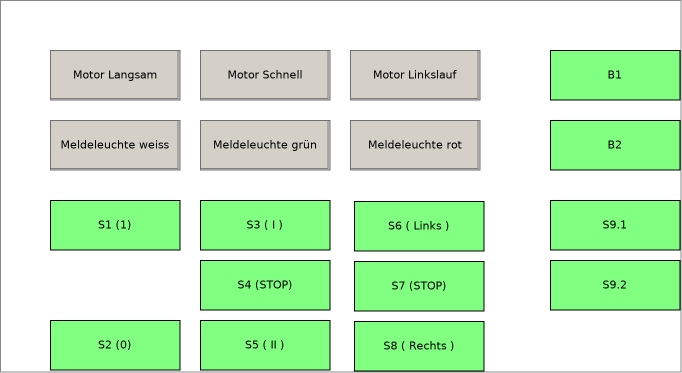
VISUALIZATION VisuGetriebemotor  // 682x373
    Button (50,50 130x50), "Motor Langsam"
        tap dSub.Q3
    Button (200,50 130x50), "Motor Schnell"
        tap dSub.Q1
    Button (350,50 130x50), "Motor Linkslauf"
        toggle dSub.Q2
    Button (50,120 130x50), "Meldeleuchte weiss"
        tap dSub.P1
    Button (200,120 130x50), "Meldeleuchte grün"
        tap dSub.P2
    Button (350,120 130x50), "Meldeleuchte rot"
        tap dSub.P3
    Rectangle (50,200 130x50), "S1 (1)", colour toggle: dSub.S1
    Rectangle (50,320 130x50), "S2 (0)", colour toggle: dSub.S2
    Rectangle (200,200 130x50), "S3 ( I )", colour toggle: dSub.S3
    Rectangle (200,260 130x50), "S4 (STOP)", colour toggle: dSub.S4
    Rectangle (200,320 130x50), "S5 ( II )", colour toggle: dSub.S5
    Rectangle (354,201 130x50), "S6 ( Links )", colour toggle: dSub.S6
    Rectangle (354,261 130x50), "S7 (STOP)", colour toggle: dSub.S7
    Rectangle (354,321 130x50), "S8 ( Rechts )", colour toggle: dSub.S8
    Rectangle (550,200 130x50), "S9.1", colour toggle: dSub.S9_1
    Rectangle (550,260 130x50), "S9.2", colour toggle: dSub.S9_2
    Rectangle (550,50 130x50), "B1", colour toggle: dSub.B1
    Rectangle (550,120 130x50), "B2", colour toggle: dSub.B2
END_VISUALIZATION

(* stored: Version 1.1.0.1, ProductVersion 3.1.4022.7
   Visu VisuGetriebemotor: Id {d2649af4-bcc3-4286-9a82-9bbb6d59b009} *)
